(* Schneider Machine Expert - Basic project 14_drum_simulation, file version 3.0.0.0 *)
(* ProjectInformations: Name=New project *)

HARDWARE
  Cpu 0: TM221C40U
  EthernetConfiguration: NetworkName=M221, IpAllocationMode=FixedAddress, IpAddress=0.0.0.0, SubnetMask=0.0.0.0
  SerialLineConfiguration: Baud=Baud19200, Parity=ParityEven, DataBits=DataBits8, StopBits=StopBits1, PhysicalMedium=PhysicalMediumRs485, TransmissionMode=TransmissionModeModbusRtu, SlaveId=1, Addressing=SlaveAddressing
  MastTask: UsePeriodScanMode=false, PeriodScan=100
  FastTask: Period=255
  CpuBehavior: StartingMode=StartAsPreviousState, AutoSaveRamOnEeprom=true, WatchdogPeriod=250

SYMBOLS  (address, symbol, comment, settings)
  %DR0        [Bits(BitForDrum(Outputs=%Q0.0), BitForDrum(Outputs=%Q0.1), BitForDrum(Outputs=%Q0.2), BitForDrum(Outputs=%Q0.3)), StepsNumber=4]

POU New POU
  (* SectionNumber=0 *)

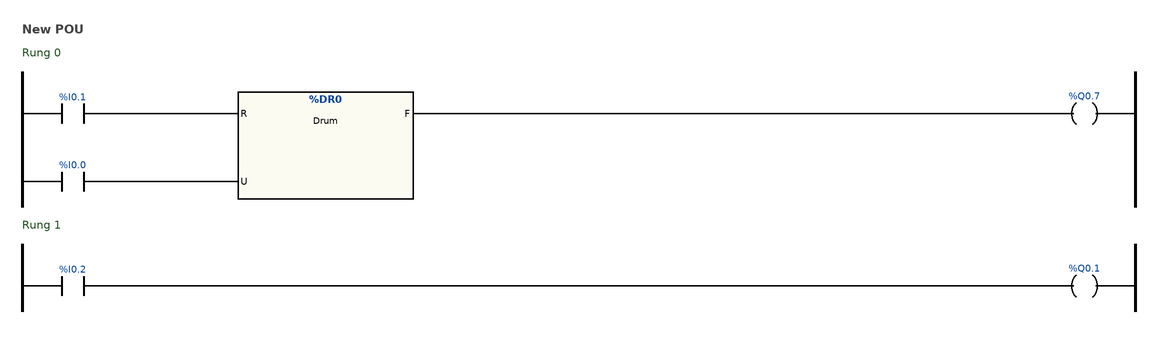

// Rung 0
  BLK %DR0
  LD %I0.1
  R
  LD %I0.0
  U
  OUT_BLK
  LD F
  ST %Q0.7
  END_BLK
  // as ST:
  //   %DR0(R := %I0.1, U := %I0.0);
  //   %Q0.7 := %DR0.F;

// Rung 1
  LD %I0.2
  ST %Q0.1
  // as ST:
  //   %Q0.1 := %I0.2;
